Fanuc KAREL source: kt00981.KL

-- PROVISIONAL review KL for V940-1; original PC SHA256 f24fa4f3a766ee8edd4f1fd125bab94b834444b9cfc9200b6f2aa85806224e45
-- Incomplete behavior may be omitted. Consult companion uncertainty JSON. Do not deploy.
PROGRAM KT00981
%NOLOCKGROUP
VAR
  I1 : INTEGER
  I2 : INTEGER
-- UNRESOLVED_DECL CFG type=00001c
-- UNRESOLVED_DECL OUT type=000106
BEGIN
  -- V9_ZERO_TABLE_METADATA_HINT layout=0001; no indexed target words; source/name/runtime held
  -- UNRESOLVED_PC offsets 5-16; opcodes 2E,23
  -- UNRESOLVED_PC offsets 21-32; opcodes 2E,23
  -- UNRESOLVED_PC offsets 37-48; opcodes 2E,23
  -- UNRESOLVED_PC offsets 53-64; opcodes 2E,23
  -- UNRESOLVED_PC offsets 69-79; opcodes 9D,22,A5
  -- UNRESOLVED_PC offsets 84-153; opcodes 27,27,21,64,27,21,64,27,21,64,27,21,64,27,21,64,27,21,64,22,76,7E,4A
  -- UNRESOLVED_PC offsets 158-162; opcodes 7F
END KT00981
